INTERFACE INTERNAL I_ReceiverNode EXTENDS I_Debug

PROPERTY INTERNAL IsOk : BOOL
GET
END_GET
END_PROPERTY

METHOD INTERNAL Receive
VAR_INPUT
	iArg			: I_Arg;
END_VAR
END_METHOD

END_INTERFACE

(* stored: Version 1.1.0.1
   Itf I_ReceiverNode: Id {8feabb5e-e1de-46c9-abdd-f60feee98617}
   Property IsOk: Id {348239b1-f517-4363-9e67-8701a65ffdfb}
   Get Get: Id {46a3294f-3f65-4ad2-8288-337eeba811e2}
   Method Receive: Id {d18b5768-d005-4abe-97ce-0acae1bb45dc} *)
